FUNCTION_BLOCK FB_Circle IMPLEMENTS I_Shape


METHOD M_Draw : BOOL
ADSLOGSTR(ADSLOG_MSGTYPE_HINT, 'Draw circle', '');
M_Draw := TRUE;
END_METHOD

END_FUNCTION_BLOCK

(* stored: Version 1.1.0.1, ProductVersion 3.1.4024.12
   POU FB_Circle: Id {0215dbf9-630e-4954-9413-5e7f95e5d02d}, SpecialFunc None
   Method M_Draw: Id {df589dcd-5658-42dc-9482-89bc0a40ce29} *)
